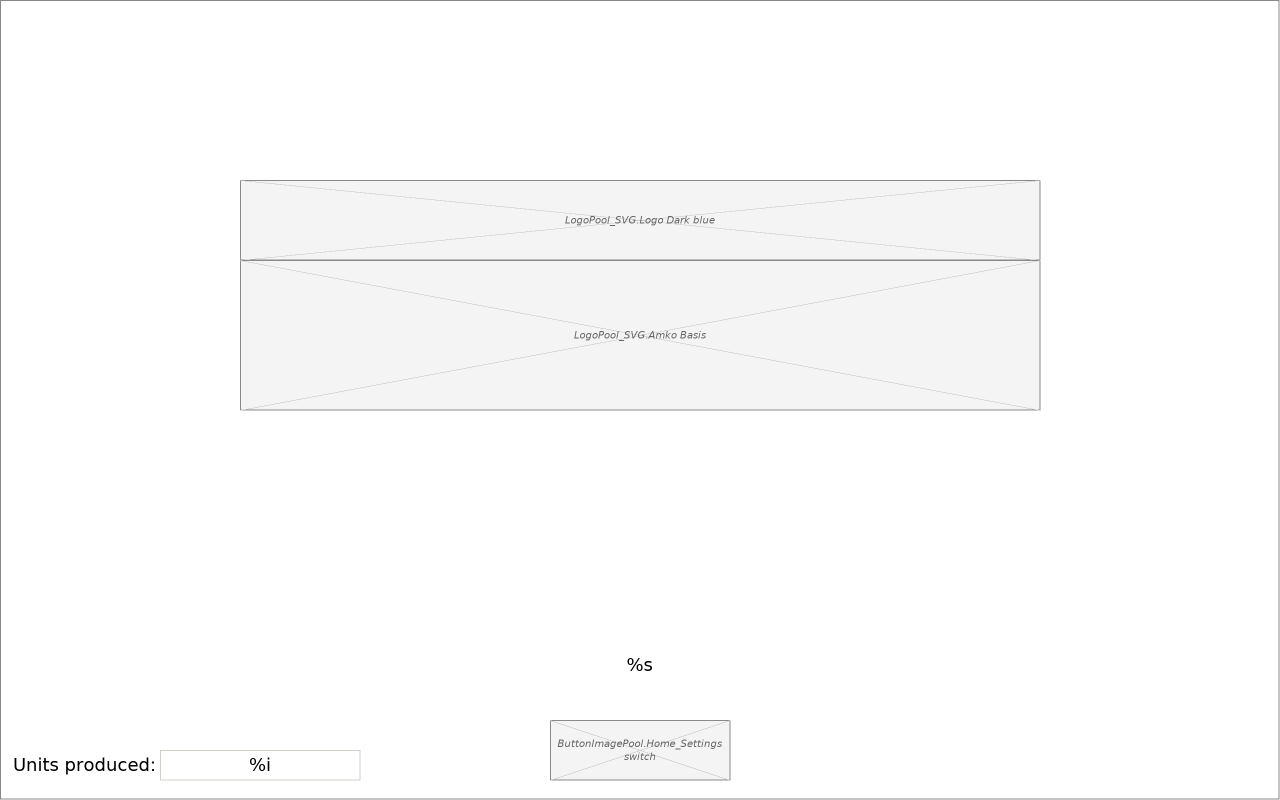
VISUALIZATION LogoScreen_SVG  // 1280x800
    Rectangle (0,0 1280x800)
    Image (240,180 800x80), image: LogoPool_SVG.Logo Dark blue
    Image (240,260 800x150), image: LogoPool_SVG.Amko Basis
    Textfield (240,650 800x30), "%s", tooltip "Operator messagages", text variable: GVL_Message.sOPeratorMessage
    Image (550,720 180x60), image: ButtonImagePool.Home_Settings switch
        OnMouseClick: execute { GVL_HMI.nStartVisu := E_StartVisu.Parameter; }
    Textfield (160,750 200x30), "%i", text variable: GVL_Main.nTotalUnitsProduced
    Label (10,750 150x30), "Units produced:"
END_VISUALIZATION

(* stored: Version 1.1.0.1, ProductVersion 3.1.4024.5
   Visu LogoScreen_SVG: Id {24a45172-ffd0-40b1-9dae-3417909fa2d0} *)
